SUBAPPLICATION Uebung_012a (* Numeric Value Input und Speichern *)
  (* Standard: 61499-2; Description: Copyright (c) 2023 Meisterschulen am Ostbahnhof This program and the accompanying materials are made available under the terms of the Eclipse Public License 2.0 which is available at https://www.eclipse.org/legal/epl-2.0/ SPDX-License-Identifier: EPL-2.0 *)
  (* Version 1.0, 2023-10-23, Franz Höpfinger, Meisterschulen am Ostbahnhof *)
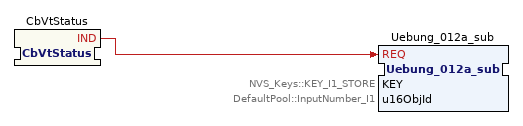
  FBS
    CbVtStatus : CbVtStatus;
  END_FBS
  SUBAPPS
    Uebung_012a_sub : Uebung_012a_sub(KEY := NVS_Keys::KEY_I1_STORE, u16ObjId := DefaultPool::InputNumber_I1);
  END_SUBAPPS
  EVENT_CONNECTIONS
    CbVtStatus.IND TO Uebung_012a_sub.REQ;
  END_CONNECTIONS
END_SUBAPPLICATION
